// TIA Portal project "SCL_blogunun_parametrelendirilmesi" (V18)

(* hardware
DEVICE "S7-1200 station_1"  S7-1200 Station
   slot 0: "Rack_0"  S7-1200 Rack  Rack  V1.0
   slot 1: "PLC_1"  CPU 1214C DC/DC/DC  6ES7 214-1AG40-0XB0  V4.6
*)

// ===== PLC "PLC_1"  CPU 1214C DC/DC/DC =====

VAR_GLOBAL   // PLC tag table "Default tag table"
   "Tag_1" AT %I0.0 : Bool;
   "Tag_2" AT %I0.1 : Bool;
   "Tag_3" AT %I0.2 : Bool;
   "Tag_4" AT %I0.3 : Bool;
   "Tag_5" AT %Q0.0 : Bool;
   "Tag_6" AT %Q0.1 : Bool;
   "Tag_7" AT %I0.4 : Bool;
   "Tag_8" AT %I0.5 : Bool;
   "Tag_9" AT %I0.6 : Bool;
   "Tag_10" AT %I0.7 : Bool;
   "Tag_11" AT %Q0.2 : Bool;
   "Tag_12" AT %Q0.3 : Bool;
END_VAR

FUNCTION "Block_1" : Void   // FC1, SCL
{ S7_Optimized_Access := 'TRUE' }
VERSION : 0.1
   VAR_INPUT
      START_1 : Bool;
      START_2 : Bool;
      START_3 : Bool;
      START_4 : Bool;
   END_VAR
   VAR_OUTPUT
      MOTOR_1 : Bool;
      MOTOR_2 : Bool;
   END_VAR
BEGIN
   #MOTOR_1 := #START_1 AND #START_2;
   #MOTOR_2 := #START_3 OR #START_4;
END_FUNCTION

ORGANIZATION_BLOCK "Main"   // OB1, LAD, ProgramCycle
TITLE = "Main Program Sweep (Cycle)"
{ S7_Optimized_Access := 'TRUE' }
VERSION : 0.1
   VAR_INPUT
      Initial_Call : Bool;   // Initial call of this OB
      Remanence : Bool;   // =True, if remanent data are available
   END_VAR
BEGIN

REGION Network 1
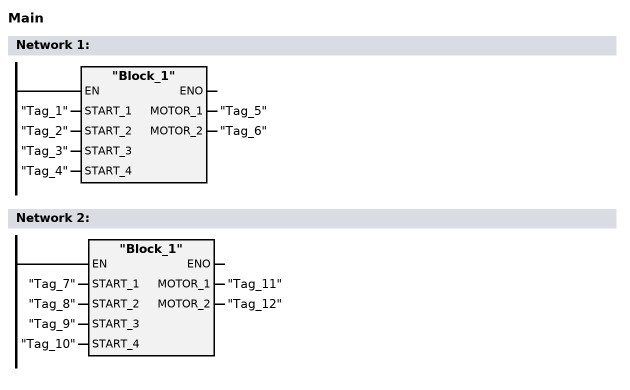
   RUNG wire#powerrail
      "Block_1"(START_1 := "Tag_1", START_2 := "Tag_2", START_3 := "Tag_3", START_4 := "Tag_4", MOTOR_1 => "Tag_5", MOTOR_2 => "Tag_6")
   END_RUNG
   // the same network as SCL:
   "Block_1"(START_1 := "Tag_1",
             START_2 := "Tag_2",
             START_3 := "Tag_3",
             START_4 := "Tag_4",
             MOTOR_1 => "Tag_5",
             MOTOR_2 => "Tag_6");
END_REGION

REGION Network 2
   RUNG wire#powerrail
      "Block_1"(START_1 := "Tag_7", START_2 := "Tag_8", START_3 := "Tag_9", START_4 := "Tag_10", MOTOR_1 => "Tag_11", MOTOR_2 => "Tag_12")
   END_RUNG
   // the same network as SCL:
   "Block_1"(START_1 := "Tag_7",
             START_2 := "Tag_8",
             START_3 := "Tag_9",
             START_4 := "Tag_10",
             MOTOR_1 => "Tag_11",
             MOTOR_2 => "Tag_12");
END_REGION
END_ORGANIZATION_BLOCK